{attribute 'GeneratedUsingTerminal: EL2522-0000-0017'}
{attribute addProperty BoxType "EL2522-0000-0017"}
{attribute addProperty Id "Set_counterBOOL1ReservedBOOL1"}
{attribute addProperty CRC "2833108354"}
{attribute addProperty Size "2"}
TYPE Control_A8DDCD82 :
STRUCT
	{attribute addProperty Name "Set_counter"}
	Set_counter : BOOL;
	{attribute addProperty Name "Reserved"}
	Reserved : BOOL;
END_STRUCT
END_TYPE

(* stored: Version 1.2.0.0, ProductVersion 3.1.4024.11
   DUT Control_A8DDCD82: Id {0d8ab03c-ed96-46e6-ace2-279b741e1e3e} *)
